PROGRAM PRG_HV_SAFETY
VAR
END_VAR

iHV_LOOP_FIM_ON:= (MR2K4_KBO_GCC_01.IG.rPRESS <= iHV_LOOP_FIM_PRESSURE) AND (MR2K4_KBO_GCC_01.IG.xPRESS_OK = TRUE);

END_PROGRAM

(* stored: Version 1.1.0.1, ProductVersion 3.1.4022.18
   POU PRG_HV_SAFETY: Id {feb92551-c00a-4a32-9bed-96e217c32cfd}, SpecialFunc None *)
